# EPICS autosave request: mcaApp/Db/Amptek_SCAn_settings.req
$(P)$(R)SCA$(N)LowChannel
$(P)$(R)SCA$(N)HighChannel
$(P)$(R)SCA$(N)OutputLevel
